INTERFACE I_Skill_Roboter

METHOD M_Reset : BOOL
VAR_INPUT
END_VAR
END_METHOD

METHOD M_Start : BOOL
VAR_INPUT
END_VAR
END_METHOD

METHOD M_Stop : BOOL
VAR_INPUT
END_VAR
END_METHOD

PROPERTY P_Prozessparameter : sRoboterProzessVariablen
SET
END_SET
END_PROPERTY

PROPERTY P_State : eSkillState
GET
END_GET
END_PROPERTY

END_INTERFACE

(* stored: Version 1.1.0.1
   Itf I_Skill_Roboter: Id {fed2c698-0a84-4171-962c-431e28adf51d}
   Method M_Reset: Id {0325ea65-64cd-4975-ba91-c2d2bdaa3263}
   Method M_Start: Id {cb1d2624-57d4-45ff-8524-3ab4c1825557}
   Method M_Stop: Id {8f0e7532-80b7-4531-ae06-4356184d7493}
   Property P_Prozessparameter: Id {d5bc063a-0693-4aae-8d75-ce595bf68605}
   Set Set: Id {03e93a44-91e9-48e3-a623-fa8d82eb39e9}
   Property P_State: Id {d1e073a8-db51-401c-ab14-ed138b30405c}
   Get Get: Id {c9e8438f-cb1e-4480-9fe3-08a3c39cb500} *)
